SUBAPPLICATION Uebung_235_AX (* Zweipunktregler (Fuellstand/Thermostat-Muster) via DualHysteresis_AR_A2X, Messwert simuliert per VT-Eingabefeld, UP/DOWN als Hintergrundfarbe auf 2 VT-Textfeldern *)
  (* Standard: 61499-2; Description: Copyright (c) 2026 Meisterschulen am Ostbahnhof This program and the accompanying materials are made available under the terms of the Eclipse Public License 2.0 which is available at https://www.eclipse.org/legal/epl-2.0/ SPDX-License-Identifier: EPL-2.0 *)
  (* Version 1.0, 2026-09-07, Franz Höpfinger, Meisterschulen am Ostbahnhof, initial API and implementation and/or initial documentation *)
  PACKAGE Uebungen;
  IMPORT Uebungen::const::UT::Dreieck::DefaultPool_Dreieck_Numeric::InputNumber_Messwert_N;
  IMPORT Uebungen::const::UT::Dreieck::DefaultPool_Dreieck::OutputString_UP;
  IMPORT Uebungen::const::UT::Dreieck::DefaultPool_Dreieck::OutputString_DOWN;
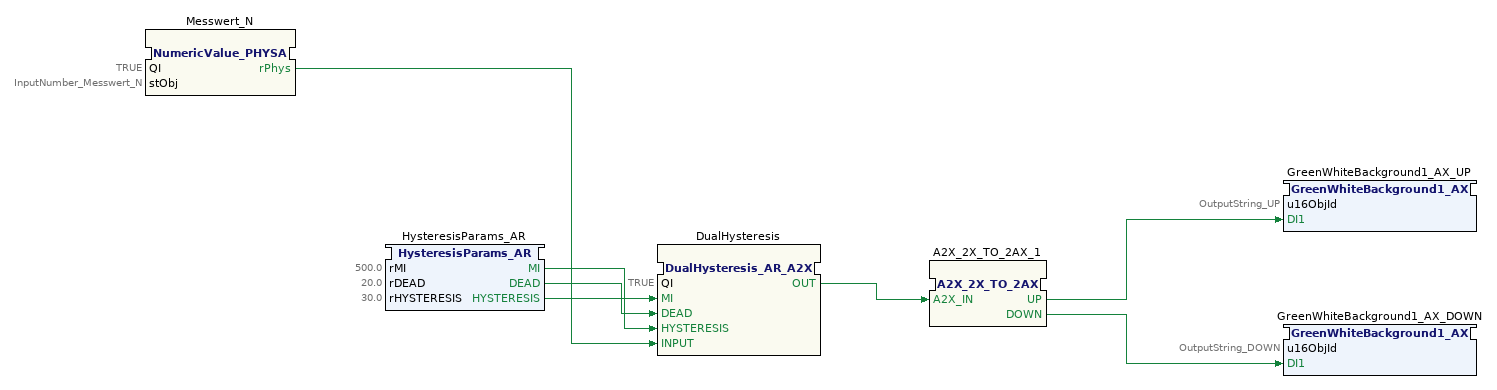
  (* Wie Uebung_234_AX, aber der Messwert kommt vom VT-Eingabefeld InputNumber_Messwert (statt echtem AI-Sensor) und UP/DOWN werden als Hintergrundfarbe von OutputString_UP/OutputString_DOWN angezeigt (statt physischer Ausgaenge). A2X_2X_TO_2AX entbuendelt UP/DOWN wieder in 2 einzelne AX-Signale, weil GreenWhiteBackground1_AX pro Instanz nur einen DI1-Eingang hat. *)
  FBS
    Messwert_N : isobus::UT::io::NumericValue::NumericValue_PHYSA(QI := TRUE, stObj := InputNumber_Messwert_N);
    DualHysteresis : logiBUS::signalprocessing::hysteresis::DualHysteresis_AR_A2X(QI := TRUE);
    A2X_2X_TO_2AX_1 : adapter::conversion::unidirectional::A2X_2X_TO_2AX;
  END_FBS
  SUBAPPS
    HysteresisParams_AR : MyLib::sys::HysteresisParams_AR(rMI := 500.0, rDEAD := 20.0, rHYSTERESIS := 30.0);
    GreenWhiteBackground1_AX_UP : MyLib::sys::GreenWhiteBackground1_AX(u16ObjId := OutputString_UP);
    GreenWhiteBackground1_AX_DOWN : MyLib::sys::GreenWhiteBackground1_AX(u16ObjId := OutputString_DOWN);
  END_SUBAPPS
  ADAPTER_CONNECTIONS
    HysteresisParams_AR.MI TO DualHysteresis.MI;
    HysteresisParams_AR.DEAD TO DualHysteresis.DEAD;
    HysteresisParams_AR.HYSTERESIS TO DualHysteresis.HYSTERESIS;
    DualHysteresis.OUT TO A2X_2X_TO_2AX_1.A2X_IN;
    A2X_2X_TO_2AX_1.UP TO GreenWhiteBackground1_AX_UP.DI1;
    A2X_2X_TO_2AX_1.DOWN TO GreenWhiteBackground1_AX_DOWN.DI1;
    Messwert_N.rPhys TO DualHysteresis.INPUT;
  END_CONNECTIONS
END_SUBAPPLICATION
